SUBAPPLICATION mapping_Buttons (* Subapplication Type *)
  (* Standard: 61499-2 *)
  (* Version 1.0, 2023-01-29, Franz *)
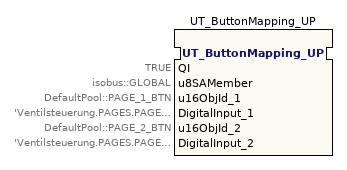
  FBS
    UT_ButtonMapping_UP : UT_ButtonMapping_UP(QI := TRUE, u8SAMember := isobus::GLOBAL, u16ObjId_1 := DefaultPool::PAGE_1_BTN, DigitalInput_1 := 'Ventilsteuerung.PAGES.PAGE_1.BTN', u16ObjId_2 := DefaultPool::PAGE_2_BTN, DigitalInput_2 := 'Ventilsteuerung.PAGES.PAGE_2.BTN');
  END_FBS
END_SUBAPPLICATION
